Fanuc KAREL source: kb00006.KL

-- PROVISIONAL review KL for V770-1; original PC SHA256 6439ee6f0f8e9ef77b14658179645df2d3b1f716cd85366ed030195d1aa12673
-- Incomplete behavior may be omitted. Consult companion uncertainty JSON. Do not deploy.
PROGRAM KB00006
%NOLOCKGROUP
BEGIN
  -- UNRESOLVED_PC offsets 5-12; opcodes 9D,23
  -- UNRESOLVED_PC offsets 17-27; opcodes 9D,22,9D,33,35
  -- UNRESOLVED_PC offsets 32-39; opcodes 9D,23
  -- UNRESOLVED_PC offsets 44-51; opcodes 9D,23
  -- UNRESOLVED_PC offsets 56-90; opcodes 27,22,22,22,22,22,31
  -- UNRESOLVED_PC offsets 95-99; opcodes 7F
END KB00006
